// TIA Portal V16 export
// export: Created 2021-09-08T12:46:15.5823651Z, ExportSetting WithDefaults, DisplayName Totally Integrated Automation Portal, DisplayVersion V16 Update 3, DisplayName TIA Portal Version Control Interface, DisplayVersion V16 Update 2, DisplayName TIA Portal Openness, DisplayVersion V16 Update 3, DisplayName TIA Portal Teamcenter Gateway, DisplayVersion V16, DisplayName STEP 7 Professional, DisplayVersion V16 Update 3, DisplayName STEP 7 Safety, DisplayVersion V16, DisplayName WinCC Advanced, DisplayVersion V16 Update 3
DATA_BLOCK "dtSetup"   // DB6
{ S7_Optimized_Access := 'FALSE' }
VERSION : 0.1
// stored: AutoNumber true, DBAccessibleFromOPCUA true, IsOnlyStoredInLoadMemory false, IsWriteProtectedInAS false
   VAR RETAIN
      workTW201 : Bool;   // 1-работа, 0-ремонт
      workTW202 : Bool;   // 1-работа, 0-ремонт
      workTW1401 : Bool;   // 1-работа, 0-ремонт
      workTW1402 : Bool;   // 1-работа, 0-ремонт
      selectTW20x : Int;
      selectTW140x : Int;
   END_VAR
BEGIN
END_DATA_BLOCK
